//==================================================================================================
//							Beckhoff Automation Poland
//								FB_AdvancedLogEvent
//									16.11.2016
//				OPIS
//  v1.2 	|| TC v 3.1.4020.28		|| - uporzadkowanie zmiennych
//  v1.1 	|| TC v 3.1.4020.0 		|| - dodanie zmiennych wejsciowych bQuitRequired, bFBCleanup, udiEventState, bQuitAck, podpiecie zmiennych Error i ErrorID
// 	v1.0 	|| TC v 3.1.4020.0 		|| - pierwsza wersja
//==================================================================================================
FUNCTION_BLOCK FB_AdvancedLogEvent
VAR_INPUT
	(*Parametry do przekazania na blok ADSLOGEVENT*)
	bSetEvent						: BOOL;
	bQuit							: BOOL;
	udiSourceID						: UDINT; 				// nr bazy
	udiEventID						: UDINT; 				// nr zdarzenia
	sFormat							: STRING;				// jak mamy parametry to wstawiamy np: %s%d jeżeli nie mamy to zostawiamy puste pole
	eEventClass						: E_TcEventClass;		// klasa błędów
	pDataAddress					: POINTER TO BYTE;		// adress zmiennych parametrów, gdy korzystamy z sFormat
	udiDataLenght					: UDINT;				// dluglosc zmiennych parametrów, gdy korzystamy sFormat
	bQuitRequired					: BOOL := FALSE;
	bFbCleanup						: BOOL := FALSE;
END_VAR
VAR_OUTPUT
	bError							: BOOL;
	udiErrorID						: UDINT;
	udiEventState					: UDINT;
	bQuitAck						: BOOL;
END_VAR
VAR
	fbLogEvent						: ADSLOGEVENT;  		// Blok wysyłający event
	Event							: TcEvent;				// Konfiguracja eventu
END_VAR

Event.bQuitRequired			:= bQuitRequired;
Event.DataFormatStrAddress	:= ADR(sFormat);
Event.StreamType			:= TCEVENTSTREAM_SIMPLE;
Event.SourceId				:= udiSourceID;
Event.Id					:= udiEventID;
Event.Class					:= eEventClass;
Event.Flags					:= TCEVENTFLAG_LOG OR TCEVENTFLAG_SRCID;
Event.ProgId				:= 'TcEventFormatter.TcXmlFormatter';

fbLogEvent(
	NETID:= , 
	PORT:= 110, 
	Event:=bSetEvent , 
	EventQuit:= bQuit, 
	EventConfigData:= Event, 
	EventDataAddress:=pDataAddress , 
	EventDataLength:=udiDataLenght , 
	FbCleanup:= bFbCleanup, 
	TMOUT:= , 
	EventState=> udiEventState, 
	Err=> bError, 
	ErrId=> udiErrorID, 
	Quit=> bQuitAck);

END_FUNCTION_BLOCK

(* stored: Version 1.1.0.1, ProductVersion 3.1.4026.13, FileIdentifier ecb02593b9089eb928a3f8015707035648100e5a, FileSignature 76db0839a0965540853dc17579a6e2c997dbef98b8b86536e11147e072c29a92988b15970002286c707817c7e2138957e3860c889d2193524d12341c38313785c38138aa72e9cacc9527c790ba1baa833981942e5ea1715394e07f06bc04452fc4c3e8f22453f8dc8b967a5814eccfcc3290815e90231581b518ff70bf7b0ca23a969af87b4f0bb21af651f3c5d254a43ea213a3ad60a8db460142eb093a232a01039a8f65273446e577bec11b565510e8f72bd9c5aa8dfb6dbcae0ec4e8856eb22b620baa9eb02cc766fed13e6f254d169e5fce6a23c3742dc7ceb38da34f8ca153b57bd2a4a0c1a27ea17d1a3f37ad22fb89a1a9492d62db9af5ff234f3aab
   POU FB_AdvancedLogEvent: Id {6fcf9ccd-87b2-497c-b619-dd932dd93596}, SpecialFunc None *)
